FUNCTION_BLOCK FB_GuidanceController IMPLEMENTS ITF_SubSystem
VAR_INPUT
	eOperationMode : GCControllerMode;
	bActive : BOOL;
	
	fDesiredDeviationFromCenterLine : REAL;
	fActualYDistance : REAL;
	fActualYAcceleration : REAL;
	fActualCurrent	: REAL;
END_VAR
VAR_OUTPUT
	fNewReferenceValueForCurrent : REAL;
	fNewRefrenceValueForForce : REAL;
	fNewreferenceValueForVoltage : REAL;
END_VAR
VAR
	//ErrorBits
	bCurrentOutOfRange : BOOL;
	bVoltageOutOfRange : BOOL;
	bForceOutOfRange	: BOOL;
END_VAR

CASE eOperationMode OF
	GCControllerMode.CurrentControlled:
		IF bActive THEN //Implement Method with Controller Structure
			doCalculateNewReferenceValueForCurrent(fDesiredDeviationFromCenterLine := fDesiredDeviationFromCenterLine,
													fActualYDistance := fActualYDistance,
													fActualYAcceleration := fActualYAcceleration,
													fActualCurrent := fActualCurrent);
		ELSE
			fNewReferenceValueForCurrent := 0;
			fNewRefrenceValueForForce := 0;
			fNewreferenceValueForVoltage := 0;
		END_IF

	GCControllerMode.ForceControlled:
		IF bActive THEN //Implement Method with Controller Structure
			doCalculateNewReferenceValueForCurrent(fDesiredDeviationFromCenterLine := fDesiredDeviationFromCenterLine,
													fActualYDistance := fActualYDistance,
													fActualYAcceleration := fActualYAcceleration,
													fActualCurrent := fActualCurrent);
		ELSE
			fNewReferenceValueForCurrent := 0;
			fNewRefrenceValueForForce := 0;	
			fNewreferenceValueForVoltage := 0;														
		END_IF
END_CASE

METHOD PRIVATE doCalculateNewReferenceValueForCurrent
VAR_INPUT
	fDesiredDeviationFromCenterLine : REAL;
	fActualYDistance : REAL;
	fActualYAcceleration : REAL;
	fActualCurrent	: REAL;
END_VAR
fNewReferenceValueForCurrent := 0;
fNewRefrenceValueForForce := 0;
fNewreferenceValueForVoltage := 0;
END_METHOD

METHOD PRIVATE doCalculateNewReferenceValueForCurrentandForce
VAR_INPUT
	fDesiredDeviationFromCenterLine : REAL;
	fActualYDistance : REAL;
	fActualYAcceleration : REAL;
	fActualCurrent	: REAL;
END_VAR
fNewReferenceValueForCurrent := 0;
fNewRefrenceValueForForce := 0;
fNewreferenceValueForVoltage := 0;
END_METHOD

PROPERTY PUBLIC eCondition : SubLevelCondition
GET
IF nErrorID <> 0 THEN
	eCondition := SubLevelCondition.ERROR;
ELSE
	eCondition := SubLevelCondition.RUN;
END_IF
END_GET
END_PROPERTY

PROPERTY PUBLIC nErrorID : UDINT
GET
//RangeAbfrage to be implemented
bCurrentOutOfRange := FALSE;
bVoltageOutOfRange := FALSE;
bForceOutOfRange := FALSE;

nErrorID.0 := bCurrentOutOfRange;
nErrorID.1 := bVoltageOutOfRange;
nErrorID.2 := bForceOutOfRange;
END_GET
END_PROPERTY

END_FUNCTION_BLOCK

(* stored: Version 1.1.0.1, ProductVersion 3.1.4024.12
   POU FB_GuidanceController: Id {b762347b-0b73-4a03-97c5-dc8d2cb401ab}, SpecialFunc None
   Method doCalculateNewReferenceValueForCurrent: Id {0266ba02-b1c4-4402-b0b0-9dcacc0680af}
   Method doCalculateNewReferenceValueForCurrentandForce: Id {0a2a5b17-8f04-42d3-8d30-42ae6c7495e1}
   Property eCondition: Id {42ce8d76-2444-4e2e-9c2b-69dafda1c213}
   Get Get: Id {5f6e61b5-784b-4549-bf76-84d3b26a008c}
   Property nErrorID: Id {d5c14b2e-f433-4c47-aa2a-9638e3371bc7}
   Get Get: Id {e3894b7e-9e1b-4973-a434-6fa91e4d3314} *)
